Yaskawa INFORM job: OK_R2_O29-32(90,0_180)OKKR.JBI

/JOB
//NAME OK_R2_O29-32(90,0_180)OKKR
///FOLDERNAME X4
//POS
///NPOS 419,419,419,25,0,0
///TOOL 0
///POSTYPE PULSE
///PULSE
C00000=97132,-107765,-123812,-202,48316,59447
C00001=96375,-92560,-98278,24892,54395,33522
C00002=118989,-99090,-96496,10423,45001,41425
C00003=119482,-98696,-96132,10013,44918,41650
C00004=120044,-95875,-95039,9417,45618,41989
C00005=120040,-96488,-95280,9446,45452,41970
C00006=120040,-96349,-93513,9613,44449,41863
C00007=116902,-102455,-99217,12157,45235,40465
C00008=92713,-84433,-91012,29057,58273,28062
C00009=92713,-84514,-90161,29225,57775,27916
C00010=92713,-84433,-91012,29057,58273,28062
C00011=94031,-81016,-89513,28080,58570,28717
C00012=92713,-84433,-91012,29057,58273,28062
C00013=90703,-81163,-89579,29929,59661,27598
C00014=92713,-84433,-91012,29057,58273,28062
C00015=92432,-93178,-97379,29384,57863,27818
C00016=124148,-115404,-96380,-35354,30522,76988
C00017=124343,-116589,-99678,-31918,27003,75506
C00018=121380,-108057,-94385,-26950,26949,73057
C00019=119584,-104006,-91933,-24006,26917,71617
C00020=119584,-103646,-90714,-24467,26399,71847
C00021=119584,-104006,-91933,-24006,26917,71617
C00022=119620,-100131,-90508,-23194,27949,71207
C00023=120534,-102543,-91401,-24964,27586,72076
C00024=122455,-107025,-93629,-28318,27362,73726
C00025=122455,-106023,-90592,-29616,26170,74375
C00026=120621,-104452,-90033,-26656,25963,72920
C00027=122455,-106023,-90592,-29616,26170,74375
C00028=124343,-116589,-99678,-31918,27003,75506
C00029=121196,-113012,-111121,-15968,43333,61367
C00030=113176,-99870,-108783,18970,68338,28733
C00031=120594,-112521,-105960,11204,51151,28139
C00032=122756,-104132,-102044,9486,52748,29227
C00033=121295,-102030,-101271,10379,53522,28693
C00034=122756,-104132,-102044,9486,52748,29227
C00035=120055,-113496,-105331,11710,50355,27811
C00036=117525,-106832,-103510,13014,52989,27048
C00037=118169,-104316,-102602,12476,53606,27398
C00038=117525,-106832,-103510,13014,52989,27048
C00039=120055,-113496,-105331,11710,50355,27811
C00040=122277,-105580,-101993,9905,52039,28956
C00041=122277,-105483,-101030,9979,51504,28904
C00042=122277,-105580,-101993,9905,52039,28956
C00043=114234,-96976,-102629,20681,62688,27649
C00044=111778,-96221,-107052,21188,70616,22267
C00045=117350,-114999,-95956,52919,38370,55080
C00046=108972,-69269,-80208,51978,72625,32902
C00047=109543,-61925,-78651,49562,78172,29234
C00048=109543,-62109,-77971,49635,77832,29052
C00049=109543,-61925,-78651,49562,78172,29234
C00050=110239,-61041,-78189,49323,77924,29446
C00051=109543,-61925,-78651,49562,78172,29234
C00052=107063,-66961,-84785,50173,80254,29118
C00053=90901,-32599,-64406,54667,92064,27755
C00054=92412,-28582,-59178,54201,90556,27610
C00055=92412,-29145,-58034,54170,89959,27242
C00056=92412,-28659,-59030,54195,90478,27561
C00057=93599,-27197,-58027,53876,89920,27837
C00058=92412,-28659,-59030,54195,90478,27561
C00059=94015,-33926,-70364,53928,92204,29442
C00060=96981,-29734,-65408,52966,90116,29668
C00061=96981,-30385,-64512,52944,89568,29346
C00062=96981,-29921,-65159,52958,89962,29578
C00063=97341,-27509,-63519,52853,89918,29730
C00064=96981,-29921,-65159,52958,89962,29578
C00065=83985,-34763,-79826,57770,100542,29760
C00066=119227,-121429,-124211,4290,80037,-5069
C00067=103198,-96938,-112022,8857,86341,-9990
C00068=104928,-94630,-110553,8370,86444,-9424
C00069=105210,-91425,-109287,8287,87275,-9277
C00070=105152,-92089,-109552,8304,87105,-9308
C00071=105152,-92773,-108542,8308,86142,-9373
C00072=104752,-96369,-111669,8420,86257,-9494
C00073=93824,-83108,-104490,-4346,83202,-15848
C00074=94227,-80625,-103370,-4481,83809,-15742
C00075=95161,-74712,-100714,-4798,85256,-15503
C00076=95037,-75505,-101078,-4756,85066,-15534
C00077=95037,-76584,-99812,-4762,83737,-15482
C00078=95852,-86288,-106522,-5052,82929,-15193
C00079=119227,-121429,-124211,4290,80037,-5069
C00080=108780,-117808,-111617,31391,23506,-27123
C00081=87227,-129275,-103249,15171,52693,-43306
C00082=62701,-112417,-81564,27325,55133,-54084
C00083=102122,-48912,-69312,5951,70900,-35879
C00084=120497,-21208,-21286,-5945,66983,-1716
C00085=120331,-15331,-14033,-5953,65534,-1703
C00086=120268,-12560,-10010,-5981,64483,-1671
C00087=120268,-12013,-7946,-6027,63500,-1622
C00088=120268,-12272,-8910,-6006,63957,-1643
C00089=120268,-12272,-8910,-6006,63957,-1643
C00090=120271,-10596,-7611,-6006,64020,-1643
C00091=120265,-13710,-11092,-5976,64558,-1676
C00092=121090,-15095,-12910,-6234,65025,-1394
C00093=122392,-36893,-37139,-6496,68816,-1124
C00094=103008,-20958,-23789,34380,46191,50944
C00095=106920,-17705,-17148,23301,36916,65920
C00096=100038,-3407,1736,8309,24573,69609
C00097=100051,-3014,2749,8424,24152,69554
C00098=100051,-2528,4297,8659,23456,69437
C00099=99986,-3534,2326,8528,24154,69501
C00100=100190,-1879,3683,8197,24147,69667
C00101=100051,-3014,2749,8424,24152,69554
C00102=107520,-15673,-12264,-3373,26664,75475
C00103=108102,-14697,-9753,25688,31788,64845
C00104=107301,-12783,-11511,23446,35942,65836
C00105=106944,-14381,-11463,24264,35264,65385
C00106=107291,-12472,-10050,14544,32367,69643
C00107=111509,-14860,-10247,839,28490,72539
C00108=99490,-13340,-18007,-5691,35272,65609
C00109=115508,-28515,-28430,-43638,36769,74115
C00110=104252,-46667,-49928,23147,42547,66097
C00111=79661,-64382,-64322,40022,51624,56449
C00112=25614,-129739,-89176,60277,72547,35569
C00113=79661,-64382,-64322,40022,51624,56449
C00114=120757,-91510,-125291,-13460,57469,-62186
C00115=120699,-18778,-86977,-11996,70937,-63715
C00116=120626,-71428,-80514,-17274,40782,-59546
C00117=119608,-71223,-77796,-25261,41295,-55541
C00118=120321,-65750,-73871,-25710,41869,-55336
C00119=120629,-71631,-77769,-17920,39069,-59168
C00120=120359,-74344,-77822,-18174,37713,-59000
C00121=130431,-63161,-72354,-39064,48875,-48581
C00122=130047,-62734,-72132,-38767,48771,-48743
C00123=122841,-56319,-67941,-39645,48811,-50497
C00124=119025,-61972,-83652,-25821,56823,-82211
C00125=119200,-79046,-90724,-17013,50162,-51422
C00126=120627,-71422,-82568,22551,39281,72893
C00127=120626,-71781,-79821,23470,37548,72366
C00128=121823,-70522,-78774,22218,37226,72958
C00129=120359,-74605,-80000,24468,36394,71829
C00130=120633,-71786,-79901,23439,37590,72383
C00131=121129,-70322,-78798,22865,37495,72644
C00132=120627,-71746,-82478,22655,39075,72833
C00133=120628,-68509,-91693,24468,73270,29259
C00134=120628,-69110,-90711,24576,72437,29080
C00135=121977,-68572,-88387,24097,71022,29276
C00136=120635,-69084,-90779,24566,72485,29092
C00137=120360,-72648,-91234,24892,71146,28701
C00138=102861,-55262,-81540,31896,79351,24316
C00139=98601,-51104,-79214,33447,81469,23349
C00140=110216,-66091,-87232,17856,68486,33346
C00141=120628,-67132,-93536,6272,76376,26037
C00142=120629,-65307,-95540,6224,78533,26146
C00143=125976,-49581,-89047,-24033,107700,27220
C00144=114932,-69047,-98963,-12803,96211,16970
C00145=121913,-67019,-96424,-19539,98441,21657
C00146=120636,-64508,-96476,-19357,99419,21079
C00147=115636,-66806,-97970,-12989,96839,17125
C00148=122528,-41117,-84074,-14839,102396,18637
C00149=119463,-45526,-86630,-11002,99586,14178
C00150=123247,-59553,-98781,-12453,98224,12183
C00151=120629,-65231,-95763,-5470,82909,26902
C00152=114225,-78059,-113057,-2895,86652,24852
C00153=100902,-64627,-95050,11985,78171,15678
C00154=98861,-75542,-94548,15732,66869,13224
C00155=119874,-71154,-93232,-19306,73218,-3187
C00156=121912,-70007,-92672,-20214,73908,-2597
C00157=98680,-77069,-90223,16254,63590,12696
C00158=96345,-50788,-86680,18048,88539,14542
C00159=93223,-76561,-100164,23339,71866,11449
C00160=120630,-61713,-98239,7195,94993,-11495
C00161=120629,-64150,-96408,7165,92633,-11631
C00162=127375,-45154,-88676,4909,106126,-9193
C00163=120636,-64104,-96466,7164,92690,-11625
C00164=119876,-67808,-97008,7371,91195,-11945
C00165=122268,-40179,-85765,5907,107177,-10698
C00166=117984,-41448,-85856,6781,104340,-12121
C00167=117785,-40415,-85699,6838,104785,-12155
C00168=118921,-47757,-88901,6950,100752,-11907
C00169=128083,-66216,-96645,288,90786,-4689
C00170=127344,-66265,-96731,512,90816,-4915
C00171=120629,-63706,-96407,7167,92858,-11618
C00172=119771,-61779,-98541,7450,95212,-11740
C00173=113204,-65987,-111954,20711,103856,62714
C00174=120630,-56479,-101004,18441,100644,64439
C00175=137486,-73235,-107371,-679,89776,64635
C00176=119374,-56629,-99297,18722,99813,63925
C00177=120637,-56952,-100808,18413,100297,64387
C00178=140905,-46902,-93805,-1895,95002,65571
C00179=144137,-98218,-105485,-6505,55837,67317
C00180=126129,-101623,-112002,18280,57665,60270
C00181=107171,-88917,-111068,40561,70673,56675
C00182=99343,-43314,-99502,42439,86261,59904
C00183=52791,5163,-64646,46831,92051,59410
C00184=-3643,-76224,-106676,-19950,71810,-76872
C00185=31759,-97415,-96886,14116,45711,-48381
C00186=44548,-99394,-97233,12419,44266,-52870
C00187=91182,-106612,-98498,6229,38996,-69241
C00188=120252,-111112,-99286,2370,35711,-79446
C00189=120252,-111112,-99286,2370,35711,-79446
C00190=122061,-111349,-89048,12693,25666,59648
C00191=121671,-62095,-66353,9610,36862,61269
C00192=121347,-21258,-21397,11816,30334,60091
C00193=120891,-15529,-14207,12963,28955,59505
C00194=120717,-13203,-11253,13455,28377,59255
C00195=120568,-11431,-9889,13625,28472,59171
C00196=120717,-13203,-11253,13455,28377,59255
C00197=120696,-12930,-10087,13737,27819,59112
C00198=120692,-12567,-8711,14046,27176,58956
C00199=120696,-12930,-10087,13737,27819,59112
C00200=120870,-15275,-13061,13229,28399,59370
C00201=123043,5425,8644,60342,36239,52197
C00202=124100,9492,13843,60466,35317,52165
C00203=124100,10308,16361,61883,34747,51389
C00204=124100,9856,14983,61106,35054,51814
C00205=123861,10994,15998,61271,35185,51717
C00206=124100,9856,14983,61106,35054,51814
C00207=124895,-3553,-1899,45295,28876,55547
C00208=121324,-21046,-20294,12047,29779,59971
C00209=121671,-62095,-66353,9610,36862,61269
C00210=122061,-111349,-89048,12693,25666,59648
C00211=120249,-110580,-95500,2498,33656,-79516
C00212=120367,-55464,-65807,1899,43695,-79179
C00213=120372,-19909,-20534,2331,34109,-79427
C00214=120603,-14858,-13386,2171,32301,-79344
C00215=118432,-12836,-10242,4853,31501,-80756
C00216=118432,-12391,-8558,4969,30699,-80814
C00217=118432,-12586,-9286,4918,31044,-80789
C00218=118432,-12586,-9286,4918,31044,-80789
C00219=118451,-11211,-8225,4888,31096,-80773
C00220=120719,-12556,-10288,2076,31575,-79294
C00221=120630,-14625,-13229,2138,32324,-79327
C00222=131566,-7566,-2012,-56880,47864,-36778
C00223=127270,2858,10417,-64219,55978,-24180
C00224=127270,2872,10457,-64230,55970,-24171
C00225=127270,3275,11649,-64548,55732,-23910
C00226=127279,2816,10434,-64241,55969,-24162
C00227=127226,4202,11617,-64241,55929,-24162
C00228=127288,2760,10411,-64252,55968,-24153
C00229=139196,1750,6280,-64814,64625,-23032
C00230=119950,-29718,-27457,2865,33344,-79709
C00231=120367,-55464,-65807,1899,43695,-79179
C00232=120071,-144849,-99630,4685,18622,-80601
C00233=120101,-156003,-112174,4198,20603,-80368
C00234=118703,-129435,-118376,15737,33464,-74082
C00235=118229,-124990,-122609,18843,37087,-72450
C00236=117709,-116078,-100914,29615,27785,-74634
C00237=121884,-95901,-99968,-19866,48605,-45126
C00238=120671,-70136,-84949,-27990,60023,-38564
C00239=120478,-67274,-83298,-27761,60367,-38737
C00240=120671,-68730,-84259,-27912,60289,-38637
C00241=120481,-64965,-83246,-27119,62754,-39366
C00242=120481,-65408,-81931,-27360,61828,-39126
C00243=121686,-66768,-84557,-27809,63026,-38954
C00244=141024,-58078,-80968,-36822,71957,-33892
C00245=140832,-52974,-76512,-36762,71783,-33908
C00246=140832,-53417,-75497,-36922,71094,-33665
C00247=140832,-52974,-76512,-36762,71783,-33908
C00248=140279,-50808,-75283,-36453,71852,-34159
C00249=140832,-52974,-76512,-36762,71783,-33908
C00250=109942,-69794,-83321,14013,53448,-56252
C00251=112063,-69620,-83237,12481,53147,-55418
C00252=109971,-72059,-85461,13968,53588,-56219
C00253=110807,-74146,-92563,12442,56365,-55924
C00254=138671,-88440,-95611,-17208,48170,-52520
C00255=138671,-88615,-94297,-17448,47310,-52358
C00256=138671,-88440,-95611,-17208,48170,-52520
C00257=138502,-86929,-95389,-16910,48750,-52704
C00258=138041,-84511,-94358,-16397,49242,-52997
C00259=138502,-86929,-95389,-16910,48750,-52704
C00260=119374,-94871,-99184,14699,45596,-69062
C00261=119374,-95024,-95430,15324,43285,-69457
C00262=120961,-93958,-95008,13845,43283,-68674
C00263=119374,-95024,-95430,15324,43285,-69457
C00264=119544,-103546,-104622,14834,44490,-69166
C00265=118175,-83390,-115370,9254,78664,-2265
C00266=136131,-54129,-95643,-4560,92395,-119
C00267=136131,-54129,-95643,-4560,92395,-119
C00268=136131,-54129,-95643,-4560,92395,-119
C00269=136131,-55910,-94548,-4553,90811,-61
C00270=136131,-54129,-95643,-4560,92395,-119
C00271=118826,-50989,-93921,11407,94620,-13199
C00272=119876,-53326,-92440,11017,92423,-13086
C00273=120690,-52300,-91874,10745,92506,-12834
C00274=119876,-53326,-92440,11017,92423,-13086
C00275=118826,-50270,-94307,11422,95216,-13144
C00276=141793,-55820,-97332,-7512,93105,2300
C00277=140356,-59957,-95696,-6990,89886,2061
C00278=139743,-58912,-95151,-6779,90039,1868
C00279=140356,-59957,-95696,-6990,89886,2061
C00280=140356,-55082,-98612,-7026,94155,1823
C00281=131844,-82412,-106901,-19181,77049,-14413
C00282=121763,-121440,-108343,-34263,48676,-32319
C00283=121436,-111193,-102207,-33362,49794,-32929
C00284=120328,-103716,-97102,-32376,49958,-33559
C00285=120328,-103424,-95545,-32743,49272,-33305
C00286=120328,-103597,-96437,-32532,49662,-33450
C00287=119706,-101713,-95741,-31911,49887,-33849
C00288=120328,-103597,-96437,-32532,49662,-33450
C00289=120421,-109652,-101209,-32668,49551,-33360
C00290=120678,-119715,-107328,-33483,48463,-32809
C00291=145717,-65257,-81010,-41655,68644,-28827
C00292=145541,-64355,-79967,-41625,68428,-28817
C00293=145541,-64661,-78699,-41864,67717,-28513
C00294=145541,-64450,-79596,-41693,68217,-28727
C00295=144419,-63348,-79027,-41165,67869,-29094
C00296=145541,-64450,-79596,-41693,68217,-28727
C00297=144489,-68274,-88356,-40433,70363,-30088
C00298=140701,-65348,-85833,-38739,68695,-31071
C00299=140701,-65803,-84785,-38949,68003,-30804
C00300=140701,-65400,-85721,-38761,68620,-31042
C00301=140042,-62987,-84490,-38345,68721,-31364
C00302=140701,-65400,-85721,-38761,68620,-31042
C00303=129105,-89797,-100104,8257,42122,63791
C00304=127638,-62786,-75319,9961,40926,62941
C00305=127541,-60842,-73212,10119,40642,62858
C00306=127452,-58887,-72168,10136,41010,62858
C00307=127541,-60842,-73212,10119,40642,62858
C00308=127484,-59721,-71596,10263,40237,62779
C00309=127484,-59825,-70645,10399,39608,62699
C00310=127484,-59721,-71596,10263,40237,62779
C00311=128516,-69367,-82634,8882,41931,63486
C00312=136804,-49406,-65089,22327,37576,67328
C00313=138316,-46303,-59486,21610,35459,67573
C00314=137893,-42671,-57282,21821,36047,67500
C00315=138034,-43342,-57719,21701,35939,67550
C00316=137984,-43593,-56312,22278,35025,67233
C00317=137984,-43463,-57769,21774,35919,67515
C00318=121497,-78215,-85327,19946,40083,59616
C00319=120626,-71657,-80701,17243,40860,59361
C00320=126255,-72821,-79643,11943,38658,61920
C00321=124460,-69554,-75696,14032,38208,60874
C00322=120888,-74575,-78008,18145,37790,58814
C00323=120633,-71857,-77956,17876,39147,58988
C00324=120627,-70525,-76194,18030,38775,58902
C00325=137917,-59445,-69070,15608,36945,73075
C00326=124488,-74552,-79755,29777,39497,66170
C00327=118213,-106277,-106559,35084,42029,63565
C00328=120627,-70570,-83191,-7863,37643,-76584
C00329=120626,-71021,-80486,-8216,35764,-76386
C00330=118158,-70995,-79054,-3103,35275,-77892
C00331=120887,-73898,-80698,-8807,34458,-76086
C00332=120633,-71014,-80560,-8214,35814,-76388
C00333=120356,-70316,-78662,-5698,35500,-76663
C00334=149514,-48084,-66762,-33033,46294,-63935
C00335=157278,-37392,-60276,-38024,50614,-61740
C00336=120626,-71358,-80242,-8280,35444,-76351
C00337=120627,-70947,-82965,-7922,37313,-76550
C00338=120635,-68263,-89533,-19357,55237,-54189
C00339=120627,-69277,-87249,-27960,61590,-38909
C00340=120627,-70131,-84728,-28472,59826,-38424
C00341=119745,-63249,-82789,-26446,65626,-40301
C00342=120887,-73269,-85067,-29013,58674,-37985
C00343=120633,-70114,-84797,-28462,59873,-38435
C00344=120443,-58955,-81680,-26193,68992,-40844
C00345=137016,-48093,-75675,-33483,76149,-36536
C00346=111378,-73522,-86374,-8880,55488,-45224
C00347=108292,-90151,-101040,-6716,55677,-46453
C00348=104551,-107393,-114036,-4170,54574,-47870
C00349=131132,-52506,-88181,2999,76585,-58563
C00350=128218,-45293,-82415,5329,83476,-42261
C00351=120634,-69367,-86746,19850,61513,-61572
C00352=119352,-71200,-86390,20819,60725,-62219
C00353=123899,-45745,-81364,10434,81835,-42081
C00354=121008,-32174,-71807,8747,81057,-38580
C00355=127442,-33341,-72503,-1454,80099,-31879
C00356=133185,-27484,-76607,-10911,90885,-32661
C00357=131562,-31841,-87200,-10336,94922,-33460
C00358=120628,-67882,-90305,-8002,60955,-27137
C00359=120628,-68780,-88641,-8118,59484,-27029
C00360=119236,-67900,-87148,-7235,58894,-27506
C00361=119351,-70586,-88688,-7347,58476,-27433
C00362=121372,-71710,-89222,-8706,58421,-26669
C00363=119224,-70326,-83140,-7530,55210,-27256
C00364=118796,-48871,-84615,-7155,80182,-30422
C00365=125592,-51833,-97720,-10091,87276,-28906
C00366=113783,-56439,-81210,-15698,57996,-69309
C00367=107790,-54952,-79381,-11557,56703,-71425
C00368=114353,-24651,-67578,-22216,88591,-34265
C00369=121370,-73680,-74765,-39382,39185,-61177
C00370=120632,-71435,-74935,-37828,39854,-62032
C00371=120118,-28187,-67292,-26229,84474,-32028
C00372=128587,-20080,-59537,-35175,87786,-29069
C00373=128865,-20064,-59811,-35543,87846,-29092
C00374=131561,-17306,-57272,-36148,87642,-28446
C00375=145089,1694,-39840,-39695,86270,-25206
C00376=146893,4898,-36831,-40237,85974,-24761
C00377=152046,17466,-29664,-47680,97969,-20185
C00378=155175,14277,-38805,-49221,102130,-20939
C00379=135677,-24502,-83351,-29476,105612,-50888
C00380=120631,-49325,-102634,-14154,102303,-71085
C00381=120630,-54638,-100904,-13945,98616,-70657
C00382=113584,-76346,-107146,-6317,84515,-70332
C00383=120637,-55119,-100712,-13931,98263,-70614
C00384=121882,-54885,-99226,-14292,97671,-70180
C00385=108764,-50124,-93744,-4400,89439,-71963
C00386=118943,-66054,-91023,-22914,66824,-68735
C00387=120627,-69075,-88308,-30031,58405,-66774
C00388=120628,-67609,-91029,-29341,60528,-67400
C00389=120651,-137986,-128118,-34242,49089,-63541
C00390=120704,-83666,-109294,-28636,63184,-68115
C00391=120704,-83666,-109294,-28636,63184,-68115
C00392=122061,-111349,-89048,12693,25666,59648
C00393=121671,-62095,-66353,9610,36862,61269
C00394=120675,-12683,-10165,1101,31339,85533
C00395=117403,-15324,-8307,14516,25200,82253
C00396=120855,-14769,-11753,884,31242,85646
C00397=120680,-13066,-11724,1072,32101,85548
C00398=112323,-11343,-6734,37915,34834,56474
C00399=106064,10956,20754,72392,53526,31980
C00400=105060,15092,17806,65581,60394,35506
C00401=113952,17541,-9445,35713,50265,81352
C00402=121726,-68659,-62259,14447,23269,58731
C00403=122061,-111349,-89048,12693,25666,59648
C00404=120249,-110580,-95500,2498,33656,-79516
C00405=120367,-55464,-65807,1899,43695,-79179
C00406=120582,872,-21183,-34353,64848,-41159
C00407=118737,3229,-13565,-31170,55800,-38986
C00408=123082,18120,-5282,-37355,69796,-35066
C00409=123254,15918,-6072,-37557,69350,-34829
C00410=101475,-2654,-13916,-26601,44193,-40098
C00411=121464,26319,17015,-59547,59899,-31656
C00412=123766,25412,14900,-59558,61805,-29104
C00413=127238,18645,4929,-58482,66393,-29908
C00414=134949,-3767,-37487,-36447,81076,-35091
C00415=139267,-30752,-53917,-52477,61088,-25483
C00416=156581,-111669,-93710,-65875,62680,-14502
C00417=153491,-118067,-95704,-59271,58057,-20364
C00418=32064,-128753,-95704,-15399,77815,718
BC00000=40617,433014,1075139
BC00001=40584,403861,1075139
BC00002=40584,403861,1075139
BC00003=40584,403861,1075139
BC00004=40584,403861,1075139
BC00005=40584,403861,1075139
BC00006=40584,403861,1075139
BC00007=40584,403861,1075139
BC00008=40578,398331,1075139
BC00009=40578,398331,1075139
BC00010=40578,398331,1075139
BC00011=40578,398331,1075139
BC00012=40578,398331,1075139
BC00013=40578,398331,1075139
BC00014=40578,398331,1075139
BC00015=40578,398331,1075139
BC00016=40578,398331,1075139
BC00017=50979,403405,1075139
BC00018=50979,403405,1075139
BC00019=50979,403405,1075139
BC00020=50979,403405,1075139
BC00021=50979,403405,1075139
BC00022=50979,403405,1075139
BC00023=50979,403405,1075139
BC00024=50979,403405,1075139
BC00025=50979,403405,1075139
BC00026=50979,403405,1075139
BC00027=50979,403405,1075139
BC00028=50979,403405,1075139
BC00029=64149,404350,1075139
BC00030=97710,406758,1075139
BC00031=97710,406758,1075139
BC00032=97710,406758,1075139
BC00033=97710,406758,1075139
BC00034=97710,406758,1075139
BC00035=97710,406758,1075139
BC00036=97710,406758,1075139
BC00037=97710,406758,1075139
BC00038=97710,406758,1075139
BC00039=97710,406758,1075139
BC00040=97710,406758,1075139
BC00041=97710,406758,1075139
BC00042=97710,406758,1075139
BC00043=97710,406758,1075139
BC00044=97710,406758,1075139
BC00045=161242,402258,1075139
BC00046=161242,402258,1075139
BC00047=161242,402258,1075139
BC00048=161242,402258,1075139
BC00049=161242,402258,1075139
BC00050=161242,402258,1075139
BC00051=161242,402258,1075139
BC00052=161242,402258,1075139
BC00053=161242,402258,1075139
BC00054=161242,402258,1075139
BC00055=161242,402258,1075139
BC00056=161242,402258,1075139
BC00057=161242,402258,1075139
BC00058=161242,402258,1075139
BC00059=161242,402258,1075139
BC00060=161242,402258,1075139
BC00061=161242,402258,1075139
BC00062=161242,402258,1075139
BC00063=161242,402258,1075139
BC00064=161242,402258,1075139
BC00065=161242,402258,1075139
BC00066=272640,323388,1075139
BC00067=272640,323388,1075139
BC00068=272640,323388,1075139
BC00069=272640,323388,1075139
BC00070=272640,323388,1075139
BC00071=272640,323388,1075139
BC00072=272640,323388,1075139
BC00073=272640,323388,1075139
BC00074=272640,323388,1075139
BC00075=272640,323388,1075139
BC00076=272640,323388,1075139
BC00077=272640,323388,1075139
BC00078=272640,323388,1075139
BC00079=272640,323388,1075139
BC00080=276492,493380,1075014
BC00081=283922,504167,1074774
BC00082=283922,472269,610106
BC00083=283922,442500,176449
BC00084=272768,401937,221279
BC00085=272768,401937,221279
BC00086=272768,401937,221279
BC00087=272768,401937,221279
BC00088=272768,401937,221279
BC00089=272768,401937,221279
BC00090=272768,401937,221279
BC00091=272768,401937,221279
BC00092=272768,401937,221279
BC00093=272768,401937,221279
BC00094=262264,430112,129839
BC00095=260478,434903,114288
BC00096=260770,434120,116830
BC00097=260770,434120,116830
BC00098=260770,434120,116830
BC00099=260770,434120,116830
BC00100=260770,434120,116830
BC00101=260770,434120,116830
BC00102=260770,434120,116830
BC00103=260446,433404,106928
BC00104=260440,433120,105532
BC00105=260440,433120,105532
BC00106=253761,433604,101646
BC00107=288425,427528,102013
BC00108=263859,415323,46172
BC00109=263451,415608,47213
BC00110=260478,434903,114288
BC00111=260478,511236,114288
BC00112=260478,511236,389201
BC00113=260478,511236,1074774
BC00114=249342,495388,1075139
BC00115=249342,453123,1075139
BC00116=249342,398563,1075139
BC00117=248917,390934,1075139
BC00118=248917,390934,1075139
BC00119=248917,390934,1075139
BC00120=248917,390934,1075139
BC00121=303920,381362,1075137
BC00122=303920,381362,1075137
BC00123=301786,381211,1075137
BC00124=278542,379565,1075139
BC00125=259231,387340,1075139
BC00126=179676,419370,1075139
BC00127=178021,414148,1075139
BC00128=177359,412059,1075139
BC00129=177359,412059,1075139
BC00130=177359,412059,1075139
BC00131=105050,424644,1075135
BC00132=106169,432153,1075139
BC00133=70414,411111,1075139
BC00134=70125,405650,1075139
BC00135=70015,403520,1075136
BC00136=70010,403466,1075139
BC00137=70010,403466,1075139
BC00138=71118,403271,1075139
BC00139=71118,403271,1075139
BC00140=71118,403271,1075139
BC00141=80355,399211,1075139
BC00142=79269,404744,1075139
BC00143=47048,382463,1075139
BC00144=47048,382463,1075139
BC00145=47290,382285,1075139
BC00146=47290,382285,1075139
BC00147=47048,382463,1075139
BC00148=47048,382463,1075139
BC00149=47048,382463,1075139
BC00150=47048,382463,1075139
BC00151=54159,396526,1075139
BC00152=54159,396526,1075139
BC00153=54976,420711,1075139
BC00154=54976,420711,1075139
BC00155=54976,420711,1075139
BC00156=54976,420711,1075139
BC00157=54976,420711,1075139
BC00158=54976,420711,1075139
BC00159=54976,420711,1075139
BC00160=110288,407592,1075139
BC00161=108089,402564,1075139
BC00162=107210,400553,1075139
BC00163=107210,400553,1075139
BC00164=107210,400553,1075139
BC00165=107210,400553,1075139
BC00166=107211,400553,1075138
BC00167=107211,400553,1075138
BC00168=127529,389139,1075138
BC00169=170976,364729,1075139
BC00170=170976,364729,1075139
BC00171=172048,366632,1075139
BC00172=174247,371661,1075139
BC00173=118968,383389,1075139
BC00174=118655,382787,1075139
BC00175=118530,382546,1075139
BC00176=118530,382546,1075139
BC00177=118530,382546,1075139
BC00178=118530,382546,1075139
BC00179=118530,382546,1075139
BC00180=125398,393784,1075139
BC00181=133032,406276,1075139
BC00182=133032,406276,1075139
BC00183=133032,519057,1075139
BC00184=199448,515539,1075137
BC00185=264734,516822,320920
BC00186=270434,516725,288277
BC00187=291219,516373,169245
BC00188=304175,516153,95046
BC00189=304175,516153,95046
BC00190=164710,484597,84331
BC00191=164710,461313,84331
BC00192=164710,444335,84331
BC00193=164710,444335,84331
BC00194=164710,444335,84331
BC00195=164710,444335,84331
BC00196=164710,444335,84331
BC00197=164710,444335,84331
BC00198=164710,444335,84331
BC00199=164710,444335,84331
BC00200=164710,444335,84331
BC00201=164710,444335,84331
BC00202=164710,444335,84331
BC00203=164710,444335,84331
BC00204=164710,444335,84331
BC00205=164710,444335,84331
BC00206=164710,444335,84331
BC00207=164710,444335,84331
BC00208=164710,444335,84331
BC00209=164710,461313,84331
BC00210=164710,484597,84331
BC00211=304175,503328,95046
BC00212=304175,483605,95046
BC00213=304175,463964,95046
BC00214=304175,463964,95046
BC00215=304175,463964,95046
BC00216=304175,463964,95046
BC00217=304175,463964,95046
BC00218=304175,463964,95046
BC00219=304175,463964,95046
BC00220=304175,463964,95046
BC00221=304175,463964,95046
BC00222=304175,463964,95046
BC00223=304175,463964,95046
BC00224=304175,463964,95046
BC00225=304175,463964,95046
BC00226=304175,463964,95046
BC00227=304175,463964,95046
BC00228=304175,463964,95046
BC00229=304175,463964,95046
BC00230=304175,463964,95046
BC00231=304175,483605,95046
BC00232=304175,483605,95046
BC00233=304175,483605,1074774
BC00234=355926,467275,1075012
BC00235=369184,436893,1075073
BC00236=383719,403587,1075139
BC00237=370208,411928,1075139
BC00238=364216,415627,1075139
BC00239=364216,415627,1075139
BC00240=364216,415627,1075139
BC00241=364216,415627,1075139
BC00242=364216,415627,1075139
BC00243=364216,415627,1075139
BC00244=364216,415627,1075139
BC00245=364216,415627,1075139
BC00246=364216,415627,1075139
BC00247=364216,415627,1075139
BC00248=364216,415627,1075139
BC00249=364216,415627,1075139
BC00250=364216,415627,1075139
BC00251=364216,415627,1075139
BC00252=364216,415627,1075139
BC00253=365215,415010,1075139
BC00254=383718,403587,1075136
BC00255=383718,403587,1075136
BC00256=383718,403587,1075136
BC00257=383718,403587,1075136
BC00258=383718,403587,1075136
BC00259=383718,403587,1075136
BC00260=383719,403587,1075139
BC00261=383719,403587,1075139
BC00262=383719,403587,1075139
BC00263=383719,403587,1075139
BC00264=383719,403587,1075139
BC00265=375748,406290,1075139
BC00266=375748,406290,1075139
BC00267=375748,406290,1075139
BC00268=375748,406290,1075139
BC00269=375748,406290,1075139
BC00270=375748,406290,1075139
BC00271=375748,406290,1075139
BC00272=375748,406290,1075139
BC00273=375748,406290,1075139
BC00274=375748,406290,1075139
BC00275=375748,406290,1075139
BC00276=375748,406290,1075139
BC00277=375748,406290,1075139
BC00278=375748,406290,1075139
BC00279=375748,406290,1075139
BC00280=375748,406290,1075139
BC00281=337302,402946,1075139
BC00282=291765,398985,1075139
BC00283=291765,398985,1075139
BC00284=291765,398985,1075139
BC00285=291765,398985,1075139
BC00286=291765,398985,1075139
BC00287=291765,398985,1075139
BC00288=291765,398985,1075139
BC00289=291765,398985,1075139
BC00290=291765,398985,1075139
BC00291=291765,398985,1075139
BC00292=291765,398985,1075139
BC00293=291765,398985,1075139
BC00294=291765,398985,1075139
BC00295=291765,398985,1075139
BC00296=291765,398985,1075139
BC00297=291765,398985,1075139
BC00298=291765,398985,1075139
BC00299=291765,398985,1075139
BC00300=291765,398985,1075139
BC00301=291765,398985,1075139
BC00302=291765,398985,1075139
BC00303=187435,398313,1075139
BC00304=187435,398313,1075139
BC00305=187435,398313,1075139
BC00306=187435,398313,1075139
BC00307=187435,398313,1075139
BC00308=187435,398313,1075139
BC00309=187435,398313,1075139
BC00310=187435,398313,1075139
BC00311=187435,398313,1075139
BC00312=187435,398313,1075139
BC00313=187435,398313,1075139
BC00314=187435,398313,1075139
BC00315=187435,398313,1075139
BC00316=187435,398313,1075139
BC00317=187435,398313,1075139
BC00318=187435,398313,1075139
BC00319=187435,398313,1075139
BC00320=187765,392864,1075139
BC00321=187897,390684,1075139
BC00322=187897,390684,1075139
BC00323=187897,390684,1075139
BC00324=132877,381205,1075139
BC00325=158463,379368,1075139
BC00326=158463,379368,1075139
BC00327=158463,379368,1075139
BC00328=350739,435166,1075139
BC00329=351069,429716,1075139
BC00330=351201,427536,1075139
BC00331=351201,427536,1075139
BC00332=351201,427536,1075139
BC00333=351201,427536,1075139
BC00334=351201,427536,1075139
BC00335=351201,427536,1075139
BC00336=274262,416493,1075139
BC00337=273932,421943,1075139
BC00338=328743,421386,1075139
BC00339=363729,421030,1075139
BC00340=364059,415580,1075139
BC00341=364191,413401,1075139
BC00342=364191,413401,1075139
BC00343=364191,413401,1075139
BC00344=359489,412582,1075139
BC00345=359489,412582,1075139
BC00346=331752,406144,1075139
BC00347=331752,406144,1075139
BC00348=331752,406144,1075139
BC00349=392796,427604,1075139
BC00350=387431,422520,1075128
BC00351=386526,422985,1075139
BC00352=386526,422985,1075139
BC00353=387430,422519,1075131
BC00354=387430,422519,1075132
BC00355=387430,422519,1075132
BC00356=387430,422519,1075132
BC00357=387430,422519,1075132
BC00358=342043,445248,1075139
BC00359=340290,438816,1075139
BC00360=339589,436243,1075139
BC00361=339589,436243,1075139
BC00362=339589,436243,1075139
BC00363=339627,436235,1075139
BC00364=339632,436234,1075139
BC00365=339632,436234,1075139
BC00366=300288,447869,1075139
BC00367=300288,447869,1075139
BC00368=303425,440840,1075139
BC00369=303425,440840,1075139
BC00370=303425,440840,1075139
BC00371=303425,440840,1075139
BC00372=303425,440840,1075139
BC00373=303425,440840,1075139
BC00374=303425,440840,1075139
BC00375=303425,440840,1075139
BC00376=303425,440840,1075139
BC00377=303425,440840,1075139
BC00378=303425,440840,1075139
BC00379=315343,410242,1075139
BC00380=323838,388433,1075139
BC00381=324223,387847,1075139
BC00382=324376,387612,1075139
BC00383=324376,387612,1075139
BC00384=324376,387612,1075139
BC00385=324376,387612,1075139
BC00386=317581,399081,1075139
BC00387=312599,407412,1075139
BC00388=310277,411229,1075139
BC00389=310277,411229,1075139
BC00390=310277,518673,1075139
BC00391=310277,518673,96424
BC00392=164710,484597,84331
BC00393=164710,461313,84331
BC00394=159113,439281,110182
BC00395=158925,437709,102628
BC00396=158897,437477,101511
BC00397=158897,437477,101511
BC00398=121456,431081,101248
BC00399=119005,430643,101157
BC00400=118719,430592,101146
BC00401=151249,477617,23438
BC00402=164710,461313,84331
BC00403=164710,484597,84331
BC00404=304175,483605,95046
BC00405=304175,483605,95046
BC00406=259564,470471,13441
BC00407=253342,466863,1030
BC00408=252854,466501,17
BC00409=252854,466501,17
BC00410=252831,466568,16
BC00411=303920,489564,17
BC00412=303920,489563,17
BC00413=303919,489562,16
BC00414=292332,480056,17
BC00415=292332,480056,17
BC00416=292332,480056,17
BC00417=293326,479218,7996
BC00418=241756,521761,7996
EC00000=798156,-1296783
EC00001=798156,-1296783
EC00002=798156,-1296783
EC00003=798156,-1296783
EC00004=798156,-1296783
EC00005=798156,-1296783
EC00006=798156,-1296783
EC00007=798156,-1296783
EC00008=798156,-1296783
EC00009=798156,-1296783
EC00010=798156,-1296783
EC00011=798156,-1296783
EC00012=798156,-1296783
EC00013=798156,-1296783
EC00014=798156,-1296783
EC00015=798156,-1296783
EC00016=798156,-1296783
EC00017=798156,-1296783
EC00018=798156,-1296783
EC00019=798156,-1296783
EC00020=798156,-1296783
EC00021=798156,-1296783
EC00022=798156,-1296783
EC00023=798156,-1296783
EC00024=798156,-1296783
EC00025=798156,-1296783
EC00026=798156,-1296783
EC00027=798156,-1296783
EC00028=798156,-1296783
EC00029=798156,-1296783
EC00030=798156,-1296783
EC00031=798156,-1296783
EC00032=798156,-1296783
EC00033=798156,-1296783
EC00034=798156,-1296783
EC00035=798156,-1296783
EC00036=798156,-1296783
EC00037=798156,-1296783
EC00038=798156,-1296783
EC00039=798156,-1296783
EC00040=798156,-1296783
EC00041=798156,-1296783
EC00042=798156,-1296783
EC00043=798156,-1296783
EC00044=798156,-1296783
EC00045=798156,-1296783
EC00046=798156,-1296783
EC00047=798156,-1296783
EC00048=798156,-1296783
EC00049=798156,-1296783
EC00050=798156,-1296783
EC00051=798156,-1296783
EC00052=798156,-1296783
EC00053=798156,-1296783
EC00054=798156,-1296783
EC00055=798156,-1296783
EC00056=798156,-1296783
EC00057=798156,-1296783
EC00058=798156,-1296783
EC00059=798156,-1296783
EC00060=798156,-1296783
EC00061=798156,-1296783
EC00062=798156,-1296783
EC00063=798156,-1296783
EC00064=798156,-1296783
EC00065=798156,-1296783
EC00066=798156,-1296783
EC00067=798156,-1296783
EC00068=798156,-1296783
EC00069=798156,-1296783
EC00070=798156,-1296783
EC00071=798156,-1296783
EC00072=798156,-1296783
EC00073=798156,-1296783
EC00074=798156,-1296783
EC00075=798156,-1296783
EC00076=798156,-1296783
EC00077=798156,-1296783
EC00078=798156,-1296783
EC00079=798156,-1296783
EC00080=798156,-1296783
EC00081=798156,-1296783
EC00082=798156,-1296783
EC00083=798156,-1296783
EC00084=798156,-1296783
EC00085=798156,-1296783
EC00086=798156,-1296783
EC00087=798156,-1296783
EC00088=798156,-1296783
EC00089=798156,-1296783
EC00090=798156,-1296783
EC00091=798156,-1296783
EC00092=798156,-1296783
EC00093=798156,-1296783
EC00094=798156,-1296783
EC00095=798156,-1296783
EC00096=798156,-1296783
EC00097=798156,-1296783
EC00098=798156,-1296783
EC00099=798156,-1296783
EC00100=798156,-1296783
EC00101=798156,-1296783
EC00102=798156,-1296783
EC00103=798156,-1296783
EC00104=798156,-1296783
EC00105=798156,-1296783
EC00106=798156,-1296783
EC00107=798156,-1296783
EC00108=798154,-1296783
EC00109=798154,-1296783
EC00110=798156,-1296783
EC00111=798156,-1296783
EC00112=798156,-1296783
EC00113=798156,-1296783
EC00114=798156,-1296783
EC00115=798156,-1296783
EC00116=798156,-1296783
EC00117=798156,-1296783
EC00118=798156,-1296783
EC00119=798156,-1296783
EC00120=798156,-1296783
EC00121=798155,-1296784
EC00122=798155,-1296784
EC00123=798155,-1296784
EC00124=798156,-1296783
EC00125=798156,-1296783
EC00126=798156,-1296783
EC00127=798156,-1296783
EC00128=798156,-1296783
EC00129=798156,-1296783
EC00130=798156,-1296783
EC00131=798155,-1296784
EC00132=798156,-1296783
EC00133=798156,-1296783
EC00134=798156,-1296783
EC00135=798154,-1296784
EC00136=798156,-1296783
EC00137=798156,-1296783
EC00138=798156,-1296783
EC00139=798156,-1296783
EC00140=798156,-1296783
EC00141=798156,-1296783
EC00142=798156,-1296783
EC00143=798156,-1296783
EC00144=798156,-1296783
EC00145=798156,-1296783
EC00146=798156,-1296783
EC00147=798156,-1296783
EC00148=798156,-1296783
EC00149=798156,-1296783
EC00150=798156,-1296783
EC00151=798156,-1296783
EC00152=798156,-1296783
EC00153=798156,-1296783
EC00154=798156,-1296783
EC00155=798156,-1296783
EC00156=798156,-1296783
EC00157=798156,-1296783
EC00158=798156,-1296783
EC00159=798156,-1296783
EC00160=798156,-1296783
EC00161=798156,-1296783
EC00162=798156,-1296783
EC00163=798156,-1296783
EC00164=798156,-1296783
EC00165=798156,-1296783
EC00166=798155,-1296784
EC00167=798155,-1296784
EC00168=798155,-1296784
EC00169=798156,-1296783
EC00170=798156,-1296783
EC00171=798156,-1296783
EC00172=798156,-1296783
EC00173=798156,-1296783
EC00174=798156,-1296783
EC00175=798156,-1296783
EC00176=798156,-1296783
EC00177=798156,-1296783
EC00178=798156,-1296783
EC00179=798156,-1296783
EC00180=798156,-1296783
EC00181=798156,-1296783
EC00182=798156,-1296783
EC00183=798156,-1296783
EC00184=798156,-1296783
EC00185=888531,-1083609
EC00186=888287,-953576
EC00187=887396,-479408
EC00188=886840,-183832
EC00189=798156,-183832
EC00190=798156,-183832
EC00191=798156,-183832
EC00192=798156,-183832
EC00193=798156,-183832
EC00194=798156,-183832
EC00195=798156,-183832
EC00196=798156,-183832
EC00197=798156,-183832
EC00198=798156,-183832
EC00199=798156,-183832
EC00200=798156,-183832
EC00201=798156,-183832
EC00202=798156,-183832
EC00203=798156,-183832
EC00204=798156,-183832
EC00205=798156,-183832
EC00206=798156,-183832
EC00207=798156,-183832
EC00208=798156,-183832
EC00209=798156,-183832
EC00210=798156,-183832
EC00211=798156,-183832
EC00212=798156,-183832
EC00213=798156,-183832
EC00214=798156,-183832
EC00215=798156,-183832
EC00216=798156,-183832
EC00217=798156,-183832
EC00218=798156,-183832
EC00219=798156,-183832
EC00220=798156,-183832
EC00221=798156,-183832
EC00222=798156,-183832
EC00223=798156,-183832
EC00224=798156,-183832
EC00225=798156,-183832
EC00226=798156,-183832
EC00227=798156,-183832
EC00228=798156,-183832
EC00229=798156,-183832
EC00230=798156,-183832
EC00231=798156,-183832
EC00232=798156,-183832
EC00233=798156,-183832
EC00234=798156,-183832
EC00235=798156,-183832
EC00236=798156,-183832
EC00237=798156,-183832
EC00238=798156,-183832
EC00239=798156,-183832
EC00240=798156,-183832
EC00241=798156,-183832
EC00242=798156,-183832
EC00243=798156,-183832
EC00244=798156,-183832
EC00245=798156,-183832
EC00246=798156,-183832
EC00247=798156,-183832
EC00248=798156,-183832
EC00249=798156,-183832
EC00250=798156,-183832
EC00251=798156,-183832
EC00252=798156,-183832
EC00253=798156,-183832
EC00254=798154,-183832
EC00255=798154,-183832
EC00256=798154,-183832
EC00257=798154,-183832
EC00258=798154,-183832
EC00259=798154,-183832
EC00260=798156,-183832
EC00261=798156,-183832
EC00262=798156,-183832
EC00263=798156,-183832
EC00264=798156,-183832
EC00265=798156,-183832
EC00266=798156,-183832
EC00267=798156,-183832
EC00268=798156,-183832
EC00269=798156,-183832
EC00270=798156,-183832
EC00271=798156,-183832
EC00272=798156,-183832
EC00273=798156,-183832
EC00274=798156,-183832
EC00275=798156,-183832
EC00276=798156,-183832
EC00277=798156,-183832
EC00278=798156,-183832
EC00279=798156,-183832
EC00280=798156,-183832
EC00281=798156,-183832
EC00282=798156,-183832
EC00283=798156,-183832
EC00284=798156,-183832
EC00285=798156,-183832
EC00286=798156,-183832
EC00287=798156,-183832
EC00288=798156,-183832
EC00289=798156,-183832
EC00290=798156,-183832
EC00291=798156,-183832
EC00292=798156,-183832
EC00293=798156,-183832
EC00294=798156,-183832
EC00295=798156,-183832
EC00296=798156,-183832
EC00297=798156,-183832
EC00298=798156,-183832
EC00299=798156,-183832
EC00300=798156,-183832
EC00301=798156,-183832
EC00302=798156,-183832
EC00303=798156,-183832
EC00304=798156,-183832
EC00305=798156,-183832
EC00306=798156,-183832
EC00307=798156,-183832
EC00308=798156,-183832
EC00309=798156,-183832
EC00310=798156,-183832
EC00311=798156,-183832
EC00312=798156,-183832
EC00313=798156,-183832
EC00314=798156,-183832
EC00315=798156,-183832
EC00316=798156,-183832
EC00317=798156,-183832
EC00318=798156,-183832
EC00319=798156,-183832
EC00320=798156,-183832
EC00321=798156,-183832
EC00322=798156,-183832
EC00323=798156,-183832
EC00324=798156,-183832
EC00325=798156,-183832
EC00326=798156,-183832
EC00327=798156,-183832
EC00328=798156,-183832
EC00329=798156,-183832
EC00330=798156,-183832
EC00331=798156,-183832
EC00332=798156,-183832
EC00333=798156,-183832
EC00334=798156,-183832
EC00335=798156,-183832
EC00336=798156,-183832
EC00337=798156,-183832
EC00338=798156,-183832
EC00339=798156,-183832
EC00340=798156,-183832
EC00341=798156,-183832
EC00342=798156,-183832
EC00343=798156,-183832
EC00344=798156,-183832
EC00345=798156,-183832
EC00346=798156,-183832
EC00347=798156,-183832
EC00348=798156,-183832
EC00349=798156,-183832
EC00350=798151,-183832
EC00351=798156,-183832
EC00352=798156,-183832
EC00353=798152,-183832
EC00354=798152,-183832
EC00355=798152,-183832
EC00356=798152,-183832
EC00357=798152,-183832
EC00358=798156,-183832
EC00359=798156,-183832
EC00360=798156,-183832
EC00361=798156,-183832
EC00362=798156,-183832
EC00363=798156,-183832
EC00364=798156,-183832
EC00365=798156,-183832
EC00366=798156,-183832
EC00367=798156,-183832
EC00368=798156,-183832
EC00369=798156,-183832
EC00370=798156,-183832
EC00371=798156,-183832
EC00372=798156,-183832
EC00373=798156,-183832
EC00374=798156,-183832
EC00375=798156,-183832
EC00376=798156,-183832
EC00377=798156,-183832
EC00378=798156,-183832
EC00379=798156,-183832
EC00380=798156,-183832
EC00381=798156,-183832
EC00382=798156,-183832
EC00383=798156,-183832
EC00384=798156,-183832
EC00385=798156,-183832
EC00386=798156,-183832
EC00387=798156,-183832
EC00388=798156,-183832
EC00389=798156,-183832
EC00390=798156,-183832
EC00391=798156,-183832
EC00392=798156,-183832
EC00393=798156,-183832
EC00394=798156,-183832
EC00395=798156,-183832
EC00396=798156,-183832
EC00397=798156,-183832
EC00398=798156,-183832
EC00399=798156,-183832
EC00400=798156,-183832
EC00401=798156,-183832
EC00402=798156,-183832
EC00403=798156,-183832
EC00404=798156,-183832
EC00405=798156,-183832
EC00406=798156,-183832
EC00407=798153,-183831
EC00408=798156,-183832
EC00409=798156,-183832
EC00410=798155,-183831
EC00411=798156,-183832
EC00412=798152,-183831
EC00413=798150,-183831
EC00414=798156,-183832
EC00415=798156,-183832
EC00416=798156,-183832
EC00417=805602,-183832
EC00418=805602,-183832
///POSTYPE BASE
///RECTAN
///RCONF 0,0,0,0,1,0,0,0,0,0,0,0,0,0,0,0,0,0,0,0,0,0,0,0
P00006=2.006,1.622,-0.565,0.0000,0.0000,0.0000
P00021=0.073,2.058,-0.109,0.0000,0.0000,0.0000
P00022=2.006,1.622,-0.565,0.0000,0.0000,0.0000
///RCONF 0,0,0,0,0,0,0,0,0,0,0,0,0,0,0,0,0,0,0,0,0,0,0,0
P00023=-2.957,-4.083,2.762,0.0000,0.0000,0.0000
P00024=-1.466,-0.226,-0.419,0.0000,0.0000,0.0000
P00031=-0.170,0.039,-0.647,0.0000,0.0000,0.0000
P00032=-0.423,0.157,3.222,0.0000,0.0000,0.0000
P00033=0.854,-1.099,3.047,0.0000,0.0000,0.0000
P00035=0.390,-0.027,1.040,0.0000,0.0000,0.0000
P00036=-2.434,0.084,0.197,0.0000,0.0000,0.0000
P00037=-1.075,5.090,-3.949,0.0000,0.0000,0.0000
P00038=0.174,-1.527,-10.860,0.0000,0.0000,0.0000
P00039=-0.109,1.838,-0.266,0.0000,0.0000,0.0000
P00040=2.716,-0.016,3.014,0.0000,0.0000,0.0000
P00050=-0.123,2.174,-1.314,0.0000,0.0000,0.0000
P00051=-5.945,4.696,-10.293,0.0000,0.0000,0.0000
P00052=-0.153,5.586,-7.982,0.0000,0.0000,0.0000
P00053=0.015,-0.644,-4.942,0.0000,0.0000,0.0000
P00054=-0.184,15.039,-0.270,0.0000,0.0000,0.0000
P00059=-2.448,-6.714,-12.718,0.0000,0.0000,0.0000
P00060=1524.284,698.404,-261.973,-0.4635,36.8346,-1.2388
P00061=1211.499,975.999,-261.374,0.5148,35.2356,175.5099
P00062=1205.574,689.500,-262.704,0.5159,35.2461,175.5270
P00070=2.449,-18.318,2.615,0.0000,0.0000,0.0000
P00071=-2.048,-0.034,-9.092,0.0000,0.0000,0.0000
//INST
///DATE 2024/11/19 21:47
///ATTR SC,RW
///GROUP1 RB1,BS1
///GROUP2 ST1
NOP
'OK_r2_O29-32(90,0_180)
'-90,180
'Path S1470
SFTOF3D
MOVJ C00000 BC00000 VJ=100.00  +MOVJ EC00000 VJ=100.00
MOVJ C00001 BC00001 VJ=100.00  +MOVJ EC00001 VJ=100.00
SMOVL C00002 BC00002 V=500.0  +MOVJ EC00002
SMOVL C00003 BC00003 V=166.7  +MOVJ EC00003
SREFP 3 C00004 BC00004  +REFP EC00004
CALL JOB:SEARCH-R1-S13D
SET P059 P006
SFTON3D P059
SMOVL C00005 BC00005 V=166.7  +MOVJ EC00005
SREFP 3 C00006 BC00006  +REFP EC00006
CALL JOB:SEARCH-R1-S13D
SET P059 P006
SFTON3D P059
SMOVL C00007 BC00007 V=166.7  +MOVJ EC00007
SFTOF3D
MOVL C00008 BC00008 V=250.0  +MOVJ EC00008 VJ=100.00
SREFP 3 C00009 BC00009  +REFP EC00009
CALL JOB:SEARCH-R1-S13D
SET P021 P006
SFTON3D P021
SMOVL C00010 BC00010 V=166.7  +MOVJ EC00010
SREFP 3 C00011 BC00011  +REFP EC00011
CALL JOB:SEARCH-R1-S13D
SET P021 P006
SFTON3D P021
SMOVL C00012 BC00012 V=166.7  +MOVJ EC00012
SREFP 3 C00013 BC00013  +REFP EC00013
CALL JOB:SEARCH-R1-S13D
SET P021 P006
SFTON3D P021
SMOVL C00014 BC00014 V=166.7  +MOVJ EC00014
SFTOF3D
MOVL C00015 BC00015 V=400.0  +MOVJ EC00015 VJ=100.00
MOVL C00016 BC00016 V=1000.0  +MOVJ EC00016 VJ=100.00
MOVJ C00017 BC00017 VJ=100.00  +MOVJ EC00017 VJ=100.00
MOVL C00018 BC00018 V=166.7  +MOVJ EC00018 VJ=100.00
SMOVL C00019 BC00019 V=166.7  +MOVJ EC00019
SREFP 3 C00020 BC00020  +REFP EC00020
CALL JOB:SEARCH-R1-S13D
SET P022 P006
SFTON3D P022
SMOVL C00021 BC00021 V=166.7  +MOVJ EC00021
SREFP 3 C00022 BC00022  +REFP EC00022
CALL JOB:SEARCH-R1-S13D
SET P022 P006
SFTON3D P022
SMOVL C00023 BC00023 V=166.7  +MOVJ EC00023
SMOVL C00024 BC00024 V=250.0  +MOVJ EC00024
SMOVL C00025 BC00025 V=166.7  +MOVJ EC00025
SREFP 3 C00026 BC00026  +REFP EC00026
CALL JOB:SEARCH-R1-S13D
SET P022 P006
SFTON3D P022
SMOVL C00027 BC00027 V=250.0  +MOVJ EC00027
MOVL C00028 BC00028 V=1000.0  +MOVJ EC00028 VJ=100.00
'Path S1472
SFTOF3D
MOVJ C00029 BC00029 VJ=100.00  +MOVJ EC00029 VJ=20.00
MOVJ C00030 BC00030 VJ=100.00  +MOVJ EC00030 VJ=100.00
MOVL C00031 BC00031 V=400.0  +MOVJ EC00031 VJ=100.00
SMOVL C00032 BC00032 V=166.7  +MOVJ EC00032
SREFP 3 C00033 BC00033  +REFP EC00033
CALL JOB:SEARCH-R1-S13D
SET P023 P006
SFTON3D P023
SMOVL C00034 BC00034 V=166.7  +MOVJ EC00034
SMOVL C00035 BC00035 V=166.7  +MOVJ EC00035
SMOVL C00036 BC00036 V=166.7  +MOVJ EC00036
SREFP 3 C00037 BC00037  +REFP EC00037
CALL JOB:SEARCH-R1-S13D
SET P023 P006
SFTON3D P023
SMOVL C00038 BC00038 V=166.7  +MOVJ EC00038
SMOVL C00039 BC00039 V=250.0  +MOVJ EC00039
SMOVL C00040 BC00040 V=250.0  +MOVJ EC00040
SREFP 3 C00041 BC00041  +REFP EC00041
CALL JOB:SEARCH-R1-S13D
SET P023 P006
SFTON3D P023
SMOVL C00042 BC00042 V=250.0  +MOVJ EC00042
MOVL C00043 BC00043 V=250.0  +MOVJ EC00043 VJ=100.00
MOVL C00044 BC00044 V=500.0  +MOVJ EC00044 VJ=100.00
'Path S1473
SFTOF3D
MOVJ C00045 BC00045 VJ=40.00  +MOVJ EC00045 VJ=100.00
MOVL C00046 BC00046 V=400.0  +MOVJ EC00046 VJ=100.00
SMOVL C00047 BC00047 V=166.7  +MOVJ EC00047
SREFP 3 C00048 BC00048  +REFP EC00048
CALL JOB:SEARCH-R1-S13D
SET P024 P006
SFTON3D P024
SMOVL C00049 BC00049 V=166.7  +MOVJ EC00049
SREFP 3 C00050 BC00050  +REFP EC00050
CALL JOB:SEARCH-R1-S13D
SET P024 P006
SFTON3D P024
SMOVL C00051 BC00051 V=166.7  +MOVJ EC00051
SFTOF3D
MOVL C00052 BC00052 V=400.0  +MOVJ EC00052 VJ=100.00
SMOVL C00053 BC00053 V=666.7  +MOVJ EC00053
SMOVL C00054 BC00054 V=166.7  +MOVJ EC00054
SREFP 3 C00055 BC00055  +REFP EC00055
CALL JOB:SEARCH-R1-S13D
SET P060 P006
SFTON3D P060
SMOVL C00056 BC00056 V=166.7  +MOVJ EC00056
SREFP 3 C00057 BC00057  +REFP EC00057
CALL JOB:SEARCH-R1-S13D
SET P060 P006
SFTON3D P060
SMOVL C00058 BC00058 V=166.7  +MOVJ EC00058
SFTOF3D
SMOVL C00059 BC00059 V=500.0  +MOVJ EC00059
SMOVL C00060 BC00060 V=166.7  +MOVJ EC00060
SREFP 3 C00061 BC00061  +REFP EC00061
CALL JOB:SEARCH-R1-S13D
SET P061 P006
SFTON3D P061
SMOVL C00062 BC00062 V=166.7  +MOVJ EC00062
SREFP 3 C00063 BC00063  +REFP EC00063
CALL JOB:SEARCH-R1-S13D
SET P061 P006
SFTON3D P061
SMOVL C00064 BC00064 V=166.7  +MOVJ EC00064
MOVL C00065 BC00065 V=1000.0  +MOVJ EC00065 VJ=100.00
'Path S1466
SFTOF3D
MOVJ C00066 BC00066 VJ=100.00  +MOVJ EC00066 VJ=100.00
MOVL C00067 BC00067 V=400.0  +MOVJ EC00067 VJ=100.00
SMOVL C00068 BC00068 V=100.0  +MOVJ EC00068
SREFP 3 C00069 BC00069  +REFP EC00069
CALL JOB:SEARCH-R1-S13D
SET P038 P006
SFTON3D P038
SMOVL C00070 BC00070 V=100.0  +MOVJ EC00070
SREFP 3 C00071 BC00071  +REFP EC00071
CALL JOB:SEARCH-R1-S13D
SET P038 P006
SFTON3D P038
SMOVL C00072 BC00072 V=100.0  +MOVJ EC00072
SFTOF3D
SMOVL C00073 BC00073 V=666.7  +MOVJ EC00073
SMOVL C00074 BC00074 V=166.7  +MOVJ EC00074
SREFP 3 C00075 BC00075  +REFP EC00075
CALL JOB:SEARCH-R1-S13D
SET P062 P006
SFTON3D P062
SMOVL C00076 BC00076 V=166.7  +MOVJ EC00076
SREFP 3 C00077 BC00077  +REFP EC00077
CALL JOB:SEARCH-R1-S13D
SET P062 P006
SFTON3D P062
SMOVL C00078 BC00078 V=166.7  +MOVJ EC00078
MOVL C00079 BC00079 V=1000.0  +MOVJ EC00079 VJ=100.00
MOVJ C00080 BC00080 VJ=100.00  +MOVJ EC00080 VJ=100.00
MOVJ C00081 BC00081 VJ=100.00  +MOVJ EC00081 VJ=100.00
MOVJ C00082 BC00082 VJ=100.00  +MOVJ EC00082 VJ=20.00
MOVJ C00083 BC00083 VJ=100.00  +MOVJ EC00083 VJ=100.00
'Path S1047
SFTOF3D
MOVJ C00084 BC00084 VJ=100.00  +MOVJ EC00084 VJ=100.00
MOVL C00085 BC00085 V=400.0  +MOVJ EC00085 VJ=100.00
SMOVL C00086 BC00086 V=166.7  +MOVJ EC00086
SREFP 3 C00087 BC00087  +REFP EC00087
CALL JOB:SEARCH-R1-S13D
SET P031 P006
SFTON3D P031
SMOVL C00088 BC00088 V=166.7  +MOVJ EC00088
SMOVL C00089 BC00089 V=166.7  +MOVJ EC00089
SREFP 3 C00090 BC00090  +REFP EC00090
CALL JOB:SEARCH-R1-S13D
SET P031 P006
SFTON3D P031
SMOVL C00091 BC00091 V=166.7  +MOVJ EC00091
MOVL C00092 BC00092 V=400.0  +MOVJ EC00092 VJ=100.00
MOVJ C00093 BC00093 VJ=100.00  +MOVJ EC00093 VJ=100.00
'KAT_ZMIANA
MOVJ C00094 BC00094 VJ=100.00  +MOVJ EC00094 VJ=20.00
'-90,180
'Path W1014
SFTOF3D
SMOVL C00095 BC00095 V=400.0  +MOVJ EC00095
SMOVL C00096 BC00096 V=333.3  +MOVJ EC00096
SMOVL C00097 BC00097 V=100.0  +MOVJ EC00097
SREFP 3 C00098 BC00098  +REFP EC00098
CALL JOB:SEARCH-R1-S13D
SET P040 P006
SFTON3D P040
SMOVL C00099 BC00099 V=100.0  +MOVJ EC00099
SREFP 3 C00100 BC00100  +REFP EC00100
CALL JOB:SEARCH-R1-S13D
SET P040 P006
SFTON3D P040
SMOVL C00101 BC00101 V=166.7  +MOVJ EC00101
SMOVL C00102 BC00102 V=400.0  +MOVJ EC00102
SFTON3D P031
SMOVL C00103 BC00103 V=166.7 PL=0  +MOVJ EC00103
SREFP 1 C00104 BC00104  +REFP EC00104
SREFP 2 C00105 BC00105  +REFP EC00105
MACRO1 MJ#(0) ARGF14
ARCON
SMOVL C00106 BC00106 V=8.3  +MOVJ EC00106
SFTON3D P040
SMOVL C00107 BC00107 V=8.3  +MOVJ EC00107
SMOVL C00108 BC00108 V=8.3  +MOVJ EC00108
ARCOF
SMOVL C00109 BC00109 V=400.0  +MOVJ EC00109
SFTOF3D
MOVJ C00110 BC00110 VJ=100.00  +MOVJ EC00110 VJ=100.00
MOVJ C00111 BC00111 VJ=100.00  +MOVJ EC00111 VJ=100.00
MOVJ C00112 BC00112 VJ=100.00  +MOVJ EC00112 VJ=20.00
MOVJ C00113 BC00113 VJ=100.00  +MOVJ EC00113 VJ=100.00
MOVJ C00114 BC00114 VJ=100.00  +MOVJ EC00114 VJ=100.00
MOVJ C00115 BC00115 VJ=100.00  +MOVJ EC00115 VJ=100.00
'Path W1467
SFTOF3D
SFTON3D P038
MOVJ C00116 BC00116 VJ=100.00  +MOVJ EC00116 VJ=100.00
SMOVL C00117 BC00117 V=400.0  +MOVJ EC00117
SMOVL C00118 BC00118 V=133.3 PL=0  +MOVJ EC00118
SREFP 1 C00119 BC00119  +REFP EC00119
SREFP 2 C00120 BC00120  +REFP EC00120
MACRO1 MJ#(0) ARGF6
ARCON
SMOVL C00121 BC00121 V=8.3  +MOVJ EC00121
SFTON3D P062
SMOVL C00122 BC00122 V=8.3  +MOVJ EC00122
SMOVL C00123 BC00123 V=8.3  +MOVJ EC00123
ARCOF
SMOVL C00124 BC00124 V=400.0  +MOVJ EC00124
SFTOF3D
'Path W1473
SFTOF3D
SFTON3D P061
MOVJ C00125 BC00125 VJ=100.00  +MOVJ EC00125 VJ=20.00
MOVJ C00126 BC00126 VJ=100.00  +MOVJ EC00126 VJ=100.00
SMOVL C00127 BC00127 V=400.0  +MOVJ EC00127
SMOVL C00128 BC00128 V=133.3 PL=0  +MOVJ EC00128
SREFP 1 C00129 BC00129  +REFP EC00129
SREFP 2 C00130 BC00130  +REFP EC00130
MACRO1 MJ#(0) ARGF14
ARCON
SFTON3D P022
SMOVL C00131 BC00131 V=8.3  +MOVJ EC00131
ARCOF
SMOVL C00132 BC00132 V=333.3  +MOVJ EC00132
SFTOF3D
SFTOF3D
'Path W1474
SFTOF3D
MOVJ C00133 BC00133 VJ=15.00  +MOVJ EC00133 VJ=100.00
MOVJ C00134 BC00134 VJ=15.00  +MOVJ EC00134 VJ=100.00
SFTON3D P059
SMOVL C00135 BC00135 V=133.3 PL=0  +MOVJ EC00135
SREFP 1 C00136 BC00136  +REFP EC00136
SREFP 2 C00137 BC00137  +REFP EC00137
MACRO1 MJ#(0) ARGF14
ARCON
SFTON3D P021
SMOVL C00138 BC00138 V=8.3  +MOVJ EC00138
SMOVL C00139 BC00139 V=8.3  +MOVJ EC00139
SMOVL C00140 BC00140 V=8.3  +MOVJ EC00140
ARCOF
SMOVL C00141 BC00141 V=400.0  +MOVJ EC00141
SMOVL C00142 BC00142 V=1000.0  +MOVJ EC00142
SFTOF3D
'Path W1475
SFTOF3D
SFTON3D P023
SMOVL C00143 BC00143 V=250.0  +MOVJ EC00143
SMOVL C00144 BC00144 V=166.7  +MOVJ EC00144
SREFP 1 C00145 BC00145  +REFP EC00145
SREFP 2 C00146 BC00146  +REFP EC00146
MACRO1 MJ#(0) ARGF14
ARCON
SMOVL C00147 BC00147 V=8.3  +MOVJ EC00147
SFTON3D P021
SMOVL C00148 BC00148 V=8.3  +MOVJ EC00148
SMOVL C00149 BC00149 V=8.3  +MOVJ EC00149
ARCOF
SMOVL C00150 BC00150 V=400.0  +MOVJ EC00150
SMOVL C00151 BC00151 V=1000.0  +MOVJ EC00151
SMOVL C00152 BC00152 V=1000.0  +MOVJ EC00152
SFTOF3D
'Path W1476
SFTOF3D
SFTON3D P023
SMOVL C00153 BC00153 V=166.7  +MOVJ EC00153
SMOVL C00154 BC00154 V=100.0 PL=0  +MOVJ EC00154
SREFP 1 C00155 BC00155  +REFP EC00155
SREFP 2 C00156 BC00156  +REFP EC00156
MACRO1 MJ#(0) ARGF6
ARCON
SMOVL C00157 BC00157 V=12.5  +MOVJ EC00157
ARCOF
SMOVL C00158 BC00158 V=400.0  +MOVJ EC00158
SMOVL C00159 BC00159 V=1000.0  +MOVJ EC00159
SFTOF3D
'Path W1477
SFTOF3D
SFTON3D P024
MOVJ C00160 BC00160 VJ=100.00  +MOVJ EC00160 VJ=100.00
SMOVL C00161 BC00161 V=166.7  +MOVJ EC00161
SMOVL C00162 BC00162 V=166.7 PL=0  +MOVJ EC00162
SREFP 1 C00163 BC00163  +REFP EC00163
SREFP 2 C00164 BC00164  +REFP EC00164
MACRO1 MJ#(0) ARGF14
ARCON
SMOVL C00165 BC00165 V=8.3  +MOVJ EC00165
SMOVL C00166 BC00166 V=8.3  +MOVJ EC00166
ARCOF
SMOVL C00167 BC00167 V=8.3  +MOVJ EC00167
ARCON
SMOVL C00168 BC00168 V=8.3  +MOVJ EC00168
SFTON3D P060
SMOVL C00169 BC00169 V=8.3  +MOVJ EC00169
SMOVL C00170 BC00170 V=8.3  +MOVJ EC00170
ARCOF
SMOVL C00171 BC00171 V=400.0  +MOVJ EC00171
MOVJ C00172 BC00172 VJ=100.00  +MOVJ EC00172 VJ=20.00
SFTOF3D
'Path W1478
SFTOF3D
SFTON3D P022
MOVJ C00173 BC00173 VJ=100.00  +MOVJ EC00173 VJ=100.00
SMOVL C00174 BC00174 V=333.3  +MOVJ EC00174
SMOVL C00175 BC00175 V=133.3 PL=0  +MOVJ EC00175
SREFP 1 C00176 BC00176  +REFP EC00176
SREFP 2 C00177 BC00177  +REFP EC00177
MACRO1 MJ#(0) ARGF6
ARCON
SMOVL C00178 BC00178 V=12.5  +MOVJ EC00178
SMOVL C00179 BC00179 V=12.5  +MOVJ EC00179
ARCOF
SMOVL C00180 BC00180 V=250.0  +MOVJ EC00180
SMOVL C00181 BC00181 V=1000.0  +MOVJ EC00181
MOVJ C00182 BC00182 VJ=100.00  +MOVJ EC00182 VJ=20.00
MOVJ C00183 BC00183 VJ=100.00  +MOVJ EC00183 VJ=20.00
MOVJ C00184 BC00184 VJ=100.00  +MOVJ EC00184 VJ=20.00
CALL JOB:CLEAN-R1_KM_NEW
SFTOF3D
'KAT_ZMIANA
MOVJ C00185 BC00185 VJ=100.00  +MOVJ EC00185 VJ=20.00
MOVJ C00186 BC00186 VJ=100.00  +MOVJ EC00186 VJ=100.00
MOVJ C00187 BC00187 VJ=100.00  +MOVJ EC00187 VJ=100.00
MOVJ C00188 BC00188 VJ=100.00  +MOVJ EC00188 VJ=100.00
MOVJ C00189 BC00189 VJ=100.00  +MOVJ EC00189 VJ=100.00
'-90,0
MOVJ C00190 BC00190 VJ=100.00  +MOVJ EC00190 VJ=100.00
MOVJ C00191 BC00191 VJ=100.00  +MOVJ EC00191 VJ=100.00
'Path S1464
SFTOF3D
MOVJ C00192 BC00192 VJ=100.00  +MOVJ EC00192 VJ=100.00
MOVL C00193 BC00193 V=166.7  +MOVJ EC00193 VJ=100.00
SMOVL C00194 BC00194 V=100.0  +MOVJ EC00194
SREFP 3 C00195 BC00195  +REFP EC00195
CALL JOB:SEARCH-R1-S13D
SET P037 P006
SFTON3D P037
SMOVL C00196 BC00196 V=100.0  +MOVJ EC00196
SMOVL C00197 BC00197 V=100.0  +MOVJ EC00197
SREFP 3 C00198 BC00198  +REFP EC00198
CALL JOB:SEARCH-R1-S13D
SET P037 P006
SFTON3D P037
SMOVL C00199 BC00199 V=100.0  +MOVJ EC00199
SFTOF3D
MOVL C00200 BC00200 V=400.0  +MOVJ EC00200 VJ=100.00
SMOVL C00201 BC00201 V=250.0  +MOVJ EC00201
SMOVL C00202 BC00202 V=100.0  +MOVJ EC00202
SREFP 3 C00203 BC00203  +REFP EC00203
CALL JOB:SEARCH-R1-S13D
SET P050 P006
SFTON3D P050
SMOVL C00204 BC00204 V=100.0  +MOVJ EC00204
SREFP 3 C00205 BC00205  +REFP EC00205
CALL JOB:SEARCH-R1-S13D
SET P050 P006
SFTON3D P050
SMOVL C00206 BC00206 V=100.0  +MOVJ EC00206
SMOVL C00207 BC00207 V=250.0  +MOVJ EC00207
MOVL C00208 BC00208 V=1000.0  +MOVJ EC00208 VJ=100.00
MOVJ C00209 BC00209 VJ=100.00  +MOVJ EC00209 VJ=100.00
MOVJ C00210 BC00210 VJ=100.00  +MOVJ EC00210 VJ=100.00
MOVJ C00211 BC00211 VJ=100.00  +MOVJ EC00211 VJ=100.00
MOVJ C00212 BC00212 VJ=100.00  +MOVJ EC00212 VJ=100.00
'Path S1468
SFTOF3D
MOVJ C00213 BC00213 VJ=100.00  +MOVJ EC00213 VJ=100.00
MOVL C00214 BC00214 V=250.0  +MOVJ EC00214 VJ=100.00
SMOVL C00215 BC00215 V=166.7  +MOVJ EC00215
SREFP 3 C00216 BC00216  +REFP EC00216
CALL JOB:SEARCH-R1-S13D
SET P039 P006
SFTON3D P039
SMOVL C00217 BC00217 V=100.0  +MOVJ EC00217
SMOVL C00218 BC00218 V=100.0  +MOVJ EC00218
SREFP 3 C00219 BC00219  +REFP EC00219
CALL JOB:SEARCH-R1-S13D
SET P039 P006
SFTON3D P039
SMOVL C00220 BC00220 V=100.0  +MOVJ EC00220
SFTOF3D
MOVL C00221 BC00221 V=400.0  +MOVJ EC00221 VJ=100.00
SMOVL C00222 BC00222 V=333.3  +MOVJ EC00222
SMOVL C00223 BC00223 V=250.0  +MOVJ EC00223
SMOVL C00224 BC00224 V=100.0  +MOVJ EC00224
SREFP 3 C00225 BC00225  +REFP EC00225
CALL JOB:SEARCH-R1-S13D
SET P051 P006
SFTON3D P051
SMOVL C00226 BC00226 V=100.0  +MOVJ EC00226
SREFP 3 C00227 BC00227  +REFP EC00227
CALL JOB:SEARCH-R1-S13D
SET P051 P006
SFTON3D P051
SMOVL C00228 BC00228 V=100.0  +MOVJ EC00228
SMOVL C00229 BC00229 V=400.0  +MOVJ EC00229
MOVL C00230 BC00230 V=166.7  +MOVJ EC00230 VJ=100.00
MOVJ C00231 BC00231 VJ=100.00  +MOVJ EC00231 VJ=100.00
MOVJ C00232 BC00232 VJ=100.00  +MOVJ EC00232 VJ=100.00
MOVJ C00233 BC00233 VJ=100.00  +MOVJ EC00233 VJ=100.00
MOVJ C00234 BC00234 VJ=100.00  +MOVJ EC00234 VJ=100.00
MOVJ C00235 BC00235 VJ=100.00  +MOVJ EC00235 VJ=20.00
'Path S1445
SFTOF3D
MOVJ C00236 BC00236 VJ=100.00  +MOVJ EC00236 VJ=100.00
MOVL C00237 BC00237 V=666.7  +MOVJ EC00237 VJ=100.00
SMOVL C00238 BC00238 V=166.7  +MOVJ EC00238
SREFP 3 C00239 BC00239  +REFP EC00239
CALL JOB:SEARCH-R1-S13D
SET P070 P006
SFTON3D P070
SMOVL C00240 BC00240 V=166.7  +MOVJ EC00240
SMOVL C00241 BC00241 V=166.7  +MOVJ EC00241
SREFP 3 C00242 BC00242  +REFP EC00242
CALL JOB:SEARCH-R1-S13D
SET P070 P006
SFTON3D P070
SMOVL C00243 BC00243 V=166.7  +MOVJ EC00243
SFTOF3D
SMOVL C00244 BC00244 V=666.7  +MOVJ EC00244
SMOVL C00245 BC00245 V=166.7  +MOVJ EC00245
SREFP 3 C00246 BC00246  +REFP EC00246
CALL JOB:SEARCH-R1-S13D
SET P071 P006
SFTON3D P071
SMOVL C00247 BC00247 V=166.7  +MOVJ EC00247
SREFP 3 C00248 BC00248  +REFP EC00248
CALL JOB:SEARCH-R1-S13D
SET P071 P006
SFTON3D P071
SMOVL C00249 BC00249 V=166.7  +MOVJ EC00249
SMOVL C00250 BC00250 V=166.7  +MOVJ EC00250
SREFP 3 C00251 BC00251  +REFP EC00251
CALL JOB:SEARCH-R1-S13D
SET P071 P006
SFTON3D P071
SMOVL C00252 BC00252 V=166.7  +MOVJ EC00252
SFTOF3D
SMOVL C00253 BC00253 V=500.0  +MOVJ EC00253
SMOVL C00254 BC00254 V=166.7  +MOVJ EC00254
SREFP 3 C00255 BC00255  +REFP EC00255
CALL JOB:SEARCH-R1-S13D
SET P035 P006
SFTON3D P035
SMOVL C00256 BC00256 V=166.7  +MOVJ EC00256
SMOVL C00257 BC00257 V=166.7  +MOVJ EC00257
SREFP 3 C00258 BC00258  +REFP EC00258
CALL JOB:SEARCH-R1-S13D
SET P035 P006
SFTON3D P035
SMOVL C00259 BC00259 V=166.7  +MOVJ EC00259
SMOVL C00260 BC00260 V=166.7  +MOVJ EC00260
SMOVL C00261 BC00261 V=166.7  +MOVJ EC00261
SREFP 3 C00262 BC00262  +REFP EC00262
CALL JOB:SEARCH-R1-S13D
SET P035 P006
SFTON3D P035
SMOVL C00263 BC00263 V=166.7  +MOVJ EC00263
MOVL C00264 BC00264 V=666.7  +MOVJ EC00264 VJ=100.00
'Path S1446
SFTOF3D
MOVJ C00265 BC00265 VJ=100.00  +MOVJ EC00265 VJ=20.00
MOVJ C00266 BC00266 VJ=100.00  +MOVJ EC00266 VJ=100.00
MOVL C00267 BC00267 V=666.7  +MOVJ EC00267 VJ=100.00
SMOVL C00268 BC00268 V=166.7  +MOVJ EC00268
SREFP 3 C00269 BC00269  +REFP EC00269
CALL JOB:SEARCH-R1-S13D
SET P036 P006
SFTON3D P036
SMOVL C00270 BC00270 V=166.7  +MOVJ EC00270
SMOVL C00271 BC00271 V=166.7  +MOVJ EC00271
SMOVL C00272 BC00272 V=166.7  +MOVJ EC00272
SREFP 3 C00273 BC00273  +REFP EC00273
CALL JOB:SEARCH-R1-S13D
SET P036 P006
SFTON3D P036
SMOVL C00274 BC00274 V=166.7  +MOVJ EC00274
SMOVL C00275 BC00275 V=666.7  +MOVJ EC00275
SMOVL C00276 BC00276 V=666.7  +MOVJ EC00276
SMOVL C00277 BC00277 V=166.7  +MOVJ EC00277
SREFP 3 C00278 BC00278  +REFP EC00278
CALL JOB:SEARCH-R1-S13D
SET P036 P006
SFTON3D P036
SMOVL C00279 BC00279 V=166.7  +MOVJ EC00279
SMOVL C00280 BC00280 V=500.0  +MOVJ EC00280
'Path S1447
SFTOF3D
MOVJ C00281 BC00281 VJ=100.00  +MOVJ EC00281 VJ=20.00
MOVJ C00282 BC00282 VJ=100.00  +MOVJ EC00282 VJ=100.00
MOVL C00283 BC00283 V=500.0  +MOVJ EC00283 VJ=100.00
SMOVL C00284 BC00284 V=166.7  +MOVJ EC00284
SREFP 3 C00285 BC00285  +REFP EC00285
CALL JOB:SEARCH-R1-S13D
SET P033 P006
SFTON3D P033
SMOVL C00286 BC00286 V=166.7  +MOVJ EC00286
SREFP 3 C00287 BC00287  +REFP EC00287
CALL JOB:SEARCH-R1-S13D
SET P033 P006
SFTON3D P033
SMOVL C00288 BC00288 V=166.7  +MOVJ EC00288
MOVL C00289 BC00289 V=500.0  +MOVJ EC00289 VJ=100.00
MOVL C00290 BC00290 V=1000.0  +MOVJ EC00290 VJ=100.00
SMOVL C00291 BC00291 V=500.0  +MOVJ EC00291
'Path S1555
SFTOF3D
SMOVL C00292 BC00292 V=166.7  +MOVJ EC00292
SREFP 3 C00293 BC00293  +REFP EC00293
CALL JOB:SEARCH-R1-S13D
SET P053 P006
SFTON3D P053
SMOVL C00294 BC00294 V=166.7  +MOVJ EC00294
SREFP 3 C00295 BC00295  +REFP EC00295
CALL JOB:SEARCH-R1-S13D
SET P053 P006
SFTON3D P053
SMOVL C00296 BC00296 V=166.7  +MOVJ EC00296
SFTOF3D
SMOVL C00297 BC00297 V=1000.0  +MOVJ EC00297
SMOVL C00298 BC00298 V=166.7  +MOVJ EC00298
SREFP 3 C00299 BC00299  +REFP EC00299
CALL JOB:SEARCH-R1-S13D
SET P052 P006
SFTON3D P052
SMOVL C00300 BC00300 V=166.7  +MOVJ EC00300
SREFP 3 C00301 BC00301  +REFP EC00301
CALL JOB:SEARCH-R1-S13D
SET P052 P006
SFTON3D P052
SMOVL C00302 BC00302 V=166.7  +MOVJ EC00302
SFTOF3D
MOVJ C00303 BC00303 VJ=100.00  +MOVJ EC00303 VJ=100.00
MOVL C00304 BC00304 V=1000.0  +MOVJ EC00304 VJ=100.00
SMOVL C00305 BC00305 V=166.7  +MOVJ EC00305
SREFP 3 C00306 BC00306  +REFP EC00306
CALL JOB:SEARCH-R1-S13D
SET P032 P006
SFTON3D P032
SMOVL C00307 BC00307 V=166.7  +MOVJ EC00307
SMOVL C00308 BC00308 V=166.7  +MOVJ EC00308
SREFP 3 C00309 BC00309  +REFP EC00309
CALL JOB:SEARCH-R1-S13D
SET P032 P006
SFTON3D P032
SFTOF3D
SMOVL C00310 BC00310 V=166.7  +MOVJ EC00310
MOVL C00311 BC00311 V=666.7  +MOVJ EC00311 VJ=100.00
SMOVL C00312 BC00312 V=666.7  +MOVJ EC00312
SFTOF3D
SMOVL C00313 BC00313 V=166.7  +MOVJ EC00313
SREFP 3 C00314 BC00314  +REFP EC00314
CALL JOB:SEARCH-R1-S13D
SET P054 P006
SFTON3D P054
SMOVL C00315 BC00315 V=166.7  +MOVJ EC00315
SREFP 3 C00316 BC00316  +REFP EC00316
CALL JOB:SEARCH-R1-S13D
SET P054 P006
SFTON3D P054
SMOVL C00317 BC00317 V=166.7  +MOVJ EC00317
MOVL C00318 BC00318 V=1000.0  +MOVJ EC00318 VJ=100.00
'-90,0
'Path W1480
SFTOF3D
SFTON3D P032
MOVJ C00319 BC00319 VJ=100.00  +MOVJ EC00319 VJ=100.00
SMOVL C00320 BC00320 V=400.0  +MOVJ EC00320
SMOVL C00321 BC00321 V=166.7 PL=0  +MOVJ EC00321
SREFP 1 C00322 BC00322  +REFP EC00322
SREFP 2 C00323 BC00323  +REFP EC00323
MACRO1 MJ#(0) ARGF6
ARCON
SFTON3D P054
SMOVL C00324 BC00324 V=8.3  +MOVJ EC00324
SMOVL C00325 BC00325 V=8.3  +MOVJ EC00325
ARCOF
SFTOF3D
SMOVL C00326 BC00326 V=400.0  +MOVJ EC00326
SMOVL C00327 BC00327 V=1000.0  +MOVJ EC00327
'Path W1481
SFTOF3D
SFTON3D P035
MOVJ C00328 BC00328 VJ=100.00  +MOVJ EC00328 VJ=100.00
SMOVL C00329 BC00329 V=400.0  +MOVJ EC00329
SMOVL C00330 BC00330 V=133.3 PL=0  +MOVJ EC00330
SREFP 1 C00331 BC00331  +REFP EC00331
SREFP 2 C00332 BC00332  +REFP EC00332
MACRO1 MJ#(0) ARGF14
ARCON
SMOVL C00333 BC00333 V=8.3  +MOVJ EC00333
SFTON3D P052
SMOVL C00334 BC00334 V=8.3  +MOVJ EC00334
SMOVL C00335 BC00335 V=8.3  +MOVJ EC00335
ARCOF
SFTOF3D
SMOVL C00336 BC00336 V=400.0  +MOVJ EC00336
SMOVL C00337 BC00337 V=1000.0  +MOVJ EC00337
SFTOF3D
MOVJ C00338 BC00338 VJ=100.00  +MOVJ EC00338 VJ=100.00
'Path W1482
SFTOF3D
MOVJ C00339 BC00339 VJ=100.00  +MOVJ EC00339 VJ=100.00
SMOVL C00340 BC00340 V=400.0  +MOVJ EC00340
SFTON3D P070
SMOVL C00341 BC00341 V=133.3 PL=0  +MOVJ EC00341
SREFP 1 C00342 BC00342  +REFP EC00342
SREFP 2 C00343 BC00343  +REFP EC00343
MACRO1 MJ#(0) ARGF9
ARCON
SMOVL C00344 BC00344 V=10.8  +MOVJ EC00344
SFTON3D P071
SMOVL C00345 BC00345 V=10.3  +MOVJ EC00345
SMOVL C00346 BC00346 V=10.3  +MOVJ EC00346
ARCOF
SMOVL C00347 BC00347 V=400.0  +MOVJ EC00347
SMOVL C00348 BC00348 V=1000.0  +MOVJ EC00348
SFTOF3D
'Path W1483
SFTOF3D
SFTON3D P021
MOVJ C00349 BC00349 VJ=100.00  +MOVJ EC00349 VJ=100.00
SMOVL C00350 BC00350 V=166.7 PL=0  +MOVJ EC00350
SREFP 1 C00351 BC00351  +REFP EC00351
SREFP 2 C00352 BC00352  +REFP EC00352
MACRO1 MJ#(0) ARGF14
ARCON
SMOVL C00353 BC00353 V=8.3  +MOVJ EC00353
SMOVL C00354 BC00354 V=8.3  +MOVJ EC00354
SMOVL C00355 BC00355 V=8.3  +MOVJ EC00355
ARCOF
SMOVL C00356 BC00356 V=400.0  +MOVJ EC00356
SMOVL C00357 BC00357 V=1000.0  +MOVJ EC00357
SFTOF3D
'Path W1484
SFTOF3D
SFTON3D P036
MOVJ C00358 BC00358 VJ=100.00  +MOVJ EC00358 VJ=100.00
SMOVL C00359 BC00359 V=400.0  +MOVJ EC00359
SMOVL C00360 BC00360 V=133.3 PL=0  +MOVJ EC00360
SREFP 1 C00361 BC00361  +REFP EC00361
SREFP 2 C00362 BC00362  +REFP EC00362
MACRO1 MJ#(0) ARGF6
ARCON
SMOVL C00363 BC00363 V=12.5  +MOVJ EC00363
ARCOF
SFTOF3D
SMOVL C00364 BC00364 V=400.0  +MOVJ EC00364
SMOVL C00365 BC00365 V=1000.0  +MOVJ EC00365
SFTOF3D
'Path W1485
SFTOF3D
SFTON3D P033
MOVJ C00366 BC00366 VJ=100.00  +MOVJ EC00366 VJ=100.00
SMOVL C00367 BC00367 V=400.0  +MOVJ EC00367
SMOVL C00368 BC00368 V=133.3 PL=0  +MOVJ EC00368
SREFP 1 C00369 BC00369  +REFP EC00369
SREFP 2 C00370 BC00370  +REFP EC00370
MACRO1 MJ#(0) ARGF14
ARCON
SMOVL C00371 BC00371 V=10.0  +MOVJ EC00371
SMOVL C00372 BC00372 V=10.0  +MOVJ EC00372
ARCOF
SMOVL C00373 BC00373 V=10.8  +MOVJ EC00373
ARCON
SMOVL C00374 BC00374 V=10.0  +MOVJ EC00374
SFTON3D P053
SMOVL C00375 BC00375 V=10.0  +MOVJ EC00375
SMOVL C00376 BC00376 V=10.0  +MOVJ EC00376
ARCOF
SFTOF3D
SMOVL C00377 BC00377 V=400.0  +MOVJ EC00377
SMOVL C00378 BC00378 V=1000.0  +MOVJ EC00378
SFTOF3D
'Path W1486
SFTOF3D
SFTON3D P036
MOVJ C00379 BC00379 VJ=100.00  +MOVJ EC00379 VJ=20.00
MOVJ C00380 BC00380 VJ=100.00  +MOVJ EC00380 VJ=100.00
SMOVL C00381 BC00381 V=500.0  +MOVJ EC00381
SMOVL C00382 BC00382 V=166.7 PL=0  +MOVJ EC00382
SREFP 1 C00383 BC00383  +REFP EC00383
SREFP 2 C00384 BC00384  +REFP EC00384
MACRO1 MJ#(0) ARGF6
ARCON
SMOVL C00385 BC00385 V=10.8  +MOVJ EC00385
SMOVL C00386 BC00386 V=10.8  +MOVJ EC00386
ARCOF
SMOVL C00387 BC00387 V=400.0  +MOVJ EC00387
SMOVL C00388 BC00388 V=1000.0  +MOVJ EC00388
SFTOF3D
MOVJ C00389 BC00389 VJ=100.00  +MOVJ EC00389 VJ=100.00
MOVJ C00390 BC00390 VJ=100.00  +MOVJ EC00390 VJ=100.00
MOVJ C00391 BC00391 VJ=100.00  +MOVJ EC00391 VJ=100.00
MOVJ C00392 BC00392 VJ=100.00  +MOVJ EC00392 VJ=100.00
MOVJ C00393 BC00393 VJ=100.00  +MOVJ EC00393 VJ=100.00
'Path W1465
SFTOF3D
SFTON3D P037
SMOVL C00394 BC00394 V=400.0  +MOVJ EC00394
SMOVL C00395 BC00395 V=133.3 PL=0  +MOVJ EC00395
SREFP 1 C00396 BC00396  +REFP EC00396
SREFP 2 C00397 BC00397  +REFP EC00397
MACRO1 MJ#(0) ARGF14
ARCON
SFTON3D P050
SMOVL C00398 BC00398 V=8.3  +MOVJ EC00398
SMOVL C00399 BC00399 V=8.3  +MOVJ EC00399
ARCOF
SMOVL C00400 BC00400 V=250.0  +MOVJ EC00400
SFTOF3D
MOVJ C00401 BC00401 VJ=100.00  +MOVJ EC00401 VJ=100.00
MOVJ C00402 BC00402 VJ=100.00  +MOVJ EC00402 VJ=100.00
MOVJ C00403 BC00403 VJ=100.00  +MOVJ EC00403 VJ=100.00
MOVJ C00404 BC00404 VJ=100.00  +MOVJ EC00404 VJ=100.00
MOVJ C00405 BC00405 VJ=100.00  +MOVJ EC00405 VJ=100.00
'Path W1469
SFTOF3D
SFTON3D P039
SMOVL C00406 BC00406 V=400.0  +MOVJ EC00406
SMOVL C00407 BC00407 V=133.3 PL=0  +MOVJ EC00407
SREFP 1 C00408 BC00408  +REFP EC00408
SREFP 2 C00409 BC00409  +REFP EC00409
MACRO1 MJ#(0) ARGF14
ARCON
SFTON3D P051
SMOVL C00410 BC00410 V=8.3  +MOVJ EC00410
SMOVL C00411 BC00411 V=8.3  +MOVJ EC00411
ARCOF
SMOVL C00412 BC00412 V=83.3  +MOVJ EC00412
SMOVL C00413 BC00413 V=133.3  +MOVJ EC00413
SFTOF3D
MOVJ C00414 BC00414 VJ=100.00  +MOVJ EC00414 VJ=100.00
MOVJ C00415 BC00415 VJ=100.00  +MOVJ EC00415 VJ=100.00
MOVJ C00416 BC00416 VJ=100.00  +MOVJ EC00416 VJ=100.00
MOVJ C00417 BC00417 VJ=100.00  +MOVJ EC00417 VJ=100.00
MOVJ C00418 BC00418 VJ=100.00  +MOVJ EC00418 VJ=20.00
END
